FUNCTION_BLOCK HB_S2M
VAR_INPUT
	Dur : TIME;
END_VAR
VAR_OUTPUT
	ET : TIME;
END_VAR
VAR
	Timer : TON;
END_VAR
VAR_IN_OUT
	Counter : USINT;
END_VAR
VAR // added by the converter: edge detectors and wires of the graphical bodies
    _w1 : BOOL;
END_VAR

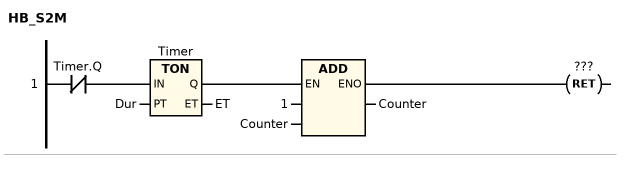
// NETWORK 1
Timer(IN := NOT Timer.Q, PT := Dur, ET => ET); // TON
_w1 := Timer.Q;
IF _w1 THEN Counter := 1 + Counter; END_IF
IF _w1 THEN RETURN; END_IF

END_FUNCTION_BLOCK

(* stored: Version 1.1.0.1, ProductVersion 3.1.4024.9
   POU HB_S2M: Id {ea62078b-64ce-4db6-8e0d-5491ab3337dc}, SpecialFunc None *)
